% RSLogix 500 project PROJECT 1 CGT PART 5.RSS, saved by version 8.30.00.16 %
PROJECT "UNTITLED"    % processor: Bul.1763 MicroLogix 1100 Series B %

PROGRAM FILES
  LAD 2 "SECTIONS"  4 rungs
  LAD 3 "INPUT"  3 rungs
  LAD 4 "LOGIC"  6 rungs
  LAD 5 "OUTPUT"  3 rungs

DATA FILES
  O0 OUTPUT  4 elements
  I1 INPUT  6 elements
  S2 STATUS  66 elements
  B3 BINARY  1 elements
  T4 TIMER  2 elements
  C5 COUNTER  1 elements
  R6 CONTROL  1 elements
  N7 INTEGER  1 elements
  F8 FLOAT  1 elements

LADDER 2 "SECTIONS"
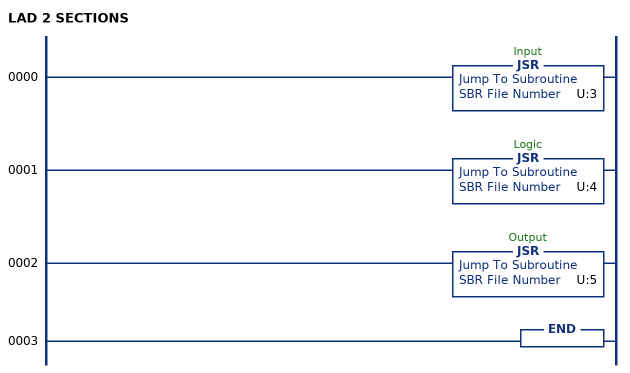
% Rung: 0 %
SOR JSR U:3 EOR
%   U:3  "Input" %
% Rung: 1 %
SOR JSR U:4 EOR
%   U:4  "Logic" %
% Rung: 2 %
SOR JSR U:5 EOR
%   U:5  "Output" %
% Rung: 3 %
SOR END EOR

LADDER 3 "INPUT"
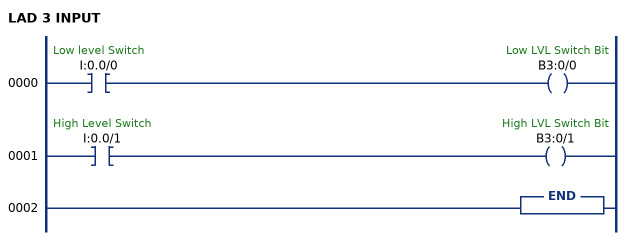
% Rung: 0 %
SOR XIC I:0.0/0 OTE B3:0/0 EOR
%   I:0.0/0  "Low level Switch" %
%   B3:0/0  "Low LVL Switch Bit" %
% Rung: 1 %
SOR XIC I:0.0/1 OTE B3:0/1 EOR
%   I:0.0/1  "High Level Switch" %
%   B3:0/1  "High LVL Switch Bit" %
% Rung: 2 %
SOR END EOR

LADDER 4 "LOGIC"
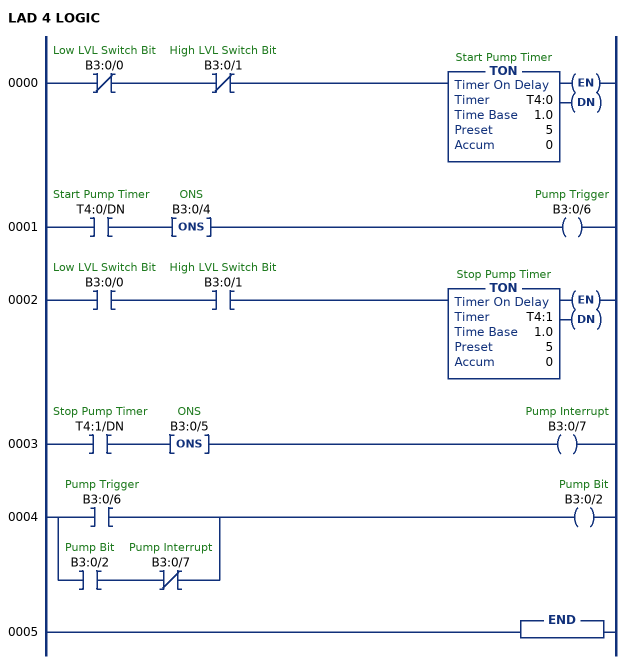
% Rung: 0 %
SOR XIO B3:0/0 XIO B3:0/1 TON T4:0 1.0 5 0 EOR
%   B3:0/0  "Low LVL Switch Bit" %
%   B3:0/1  "High LVL Switch Bit" %
%   T4:0  "Start Pump Timer" %
% Rung: 1 %
SOR XIC T4:0/DN ONS B3:0/4 OTE B3:0/6 EOR
%   T4:0  "Start Pump Timer" %
%   B3:0/4  "ONS" %
%   B3:0/6  "Pump Trigger" %
% Rung: 2 %
SOR XIC B3:0/0 XIC B3:0/1 TON T4:1 1.0 5 0 EOR
%   B3:0/0  "Low LVL Switch Bit" %
%   B3:0/1  "High LVL Switch Bit" %
%   T4:1  "Stop Pump Timer" %
% Rung: 3 %
SOR XIC T4:1/DN ONS B3:0/5 OTE B3:0/7 EOR
%   T4:1  "Stop Pump Timer" %
%   B3:0/5  "ONS" %
%   B3:0/7  "Pump Interrupt" %
% Rung: 4 %
SOR BST XIC B3:0/6 NXB XIC B3:0/2 XIO B3:0/7 BND OTE B3:0/2 EOR
%   B3:0/6  "Pump Trigger" %
%   B3:0/2  "Pump Bit" %
%   B3:0/7  "Pump Interrupt" %
% Rung: 5 %
SOR END EOR

LADDER 5 "OUTPUT"
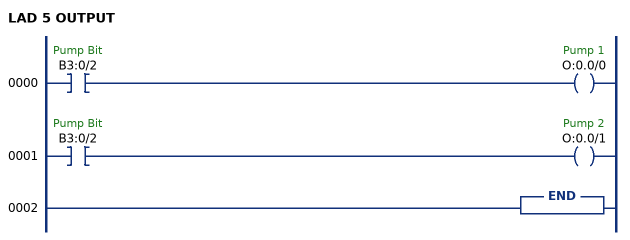
% Rung: 0 %
SOR XIC B3:0/2 OTE O:0.0/0 EOR
%   B3:0/2  "Pump Bit" %
%   O:0.0/0  "Pump 1" %
% Rung: 1 %
SOR XIC B3:0/2 OTE O:0.0/1 EOR
%   B3:0/2  "Pump Bit" %
%   O:0.0/1  "Pump 2" %
% Rung: 2 %
SOR END EOR

OTHER DOCUMENTED ADDRESSES
  B3:0/3  "Pump Bit"

DATA TABLE (non-zero values as saved)
DATA T4
% .PRE .ACC %
% T4:0 % 5 0
% T4:1 % 5 0
